FUNCTION_BLOCK SM_Torque
VAR_INPUT
	///New torque in Nm
	{attribute 'OPC.UA.DA' := '0'}
	newNewtonmeterValue: LREAL;
END_VAR
VAR_OUTPUT
	///Current status description
	{attribute 'OPC.UA.DA' := '1'}
	{attribute 'OPC.UA.DA.Access' := '1'}
	actualStatus: STRING;
	///Torque in Nm
	{attribute 'OPC.UA.DA' := '1'}
	{attribute 'OPC.UA.DA.Access' := '1'}
	newtonmeter: QuantityValue;
END_VAR
VAR_IN_OUT
END_VAR
VAR
END_VAR

newtonmeter(
    value := newNewtonmeterValue,
    unit := Units.NEWTONMETER);

END_FUNCTION_BLOCK

(* stored: Version 1.1.0.1, ProductVersion 3.1.4019.2
   POU SM_Torque: Id {9a7cde26-1cc6-4b00-8c9c-35b443f354f8}, SpecialFunc None *)
